// SIMATIC S7-200 project (STEP 7-Micro/WIN), CPU 224 REL 02.01

SYMBOL_TABLE USER1
S1               I0.0
S2               I0.1
S3               I0.2
S4               I0.3
S5               I0.4
S6               I0.5
S7               I0.6
C1S_BW           I1.2     // CY01 S1
C1S_FW           I1.1     // CY01 S2
C2S_UP           I1.0     // CY02 S1
C2S_DWN          I1.3     // CY02 S2
CNV_1            Q1.0
CNV_2            Q1.2
CNV_3            Q1.4
RODLESS          Q0.0
TN_1             Q0.1
TN_2             Q0.6
SUCTION          Q0.2
GRIPPER          Q0.5
CY_1             Q0.3
CY_2             Q0.4
END_SYMBOL_TABLE

ORGANIZATION_BLOCK MAIN:OB1
TITLE=PROGRAM COMMENTS
BEGIN
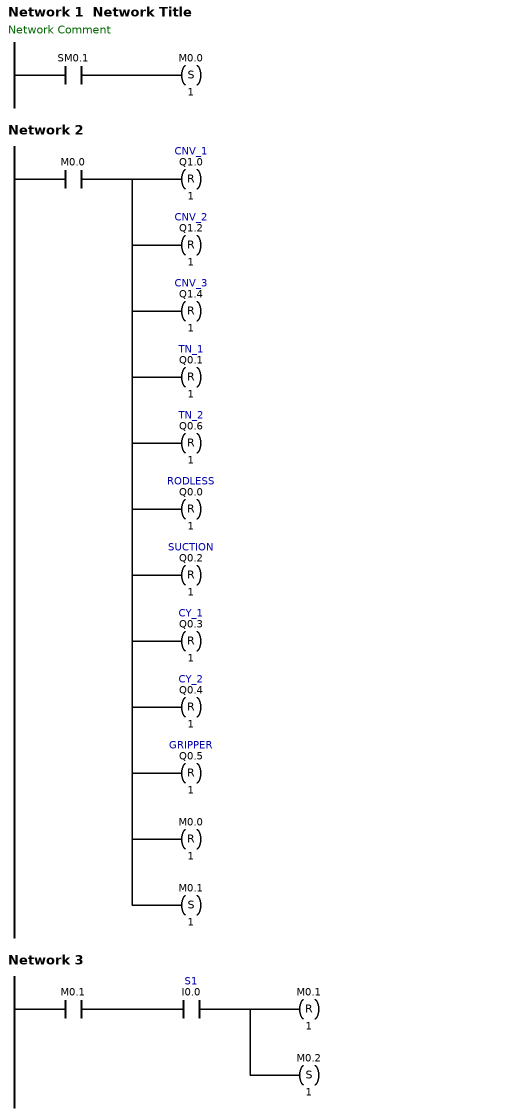
Network 1 // Network Title
// Network Comment
LD     SM0.1
S      M0.0, 1
Network 2
LD     M0.0
R      CNV_1:Q1.0, 1
R      CNV_2:Q1.2, 1
R      CNV_3:Q1.4, 1
R      TN_1:Q0.1, 1
R      TN_2:Q0.6, 1
R      RODLESS:Q0.0, 1
R      SUCTION:Q0.2, 1
R      CY_1:Q0.3, 1
R      CY_2:Q0.4, 1
R      GRIPPER:Q0.5, 1
R      M0.0, 1
S      M0.1, 1
Network 3
LD     M0.1
A      S1:I0.0
R      M0.1, 1
S      M0.2, 1
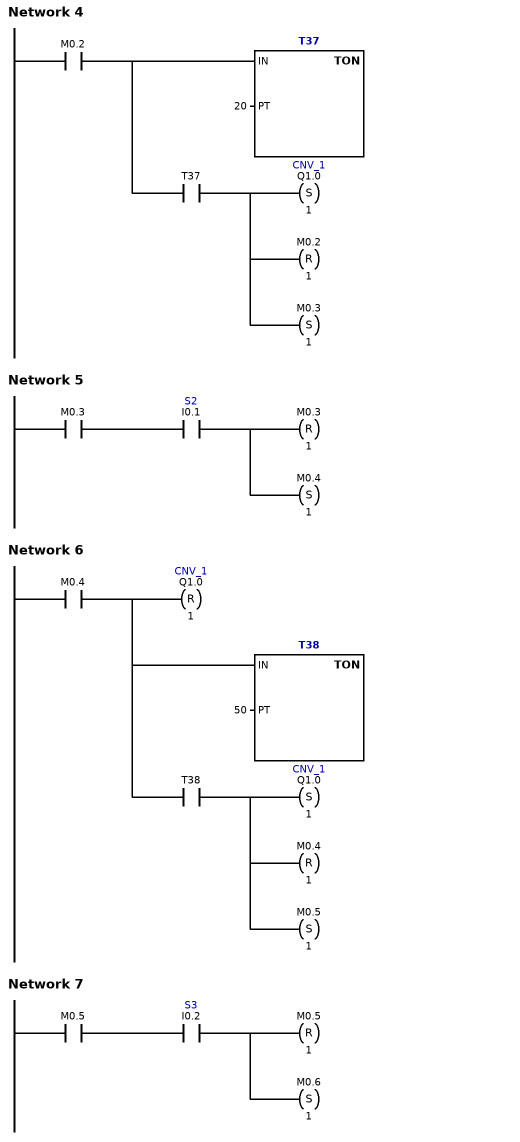
Network 4
LD     M0.2
TON    T37, 20
A      T37
S      CNV_1:Q1.0, 1
R      M0.2, 1
S      M0.3, 1
Network 5
LD     M0.3
A      S2:I0.1
R      M0.3, 1
S      M0.4, 1
Network 6
LD     M0.4
R      CNV_1:Q1.0, 1
TON    T38, 50
A      T38
S      CNV_1:Q1.0, 1
R      M0.4, 1
S      M0.5, 1
Network 7
LD     M0.5
A      S3:I0.2
R      M0.5, 1
S      M0.6, 1
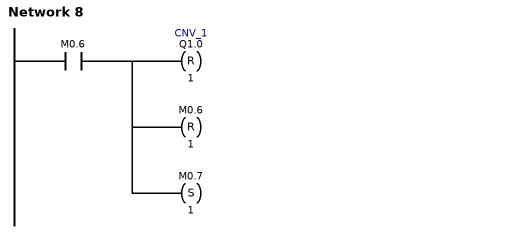
Network 8
LD     M0.6
R      CNV_1:Q1.0, 1
R      M0.6, 1
S      M0.7, 1
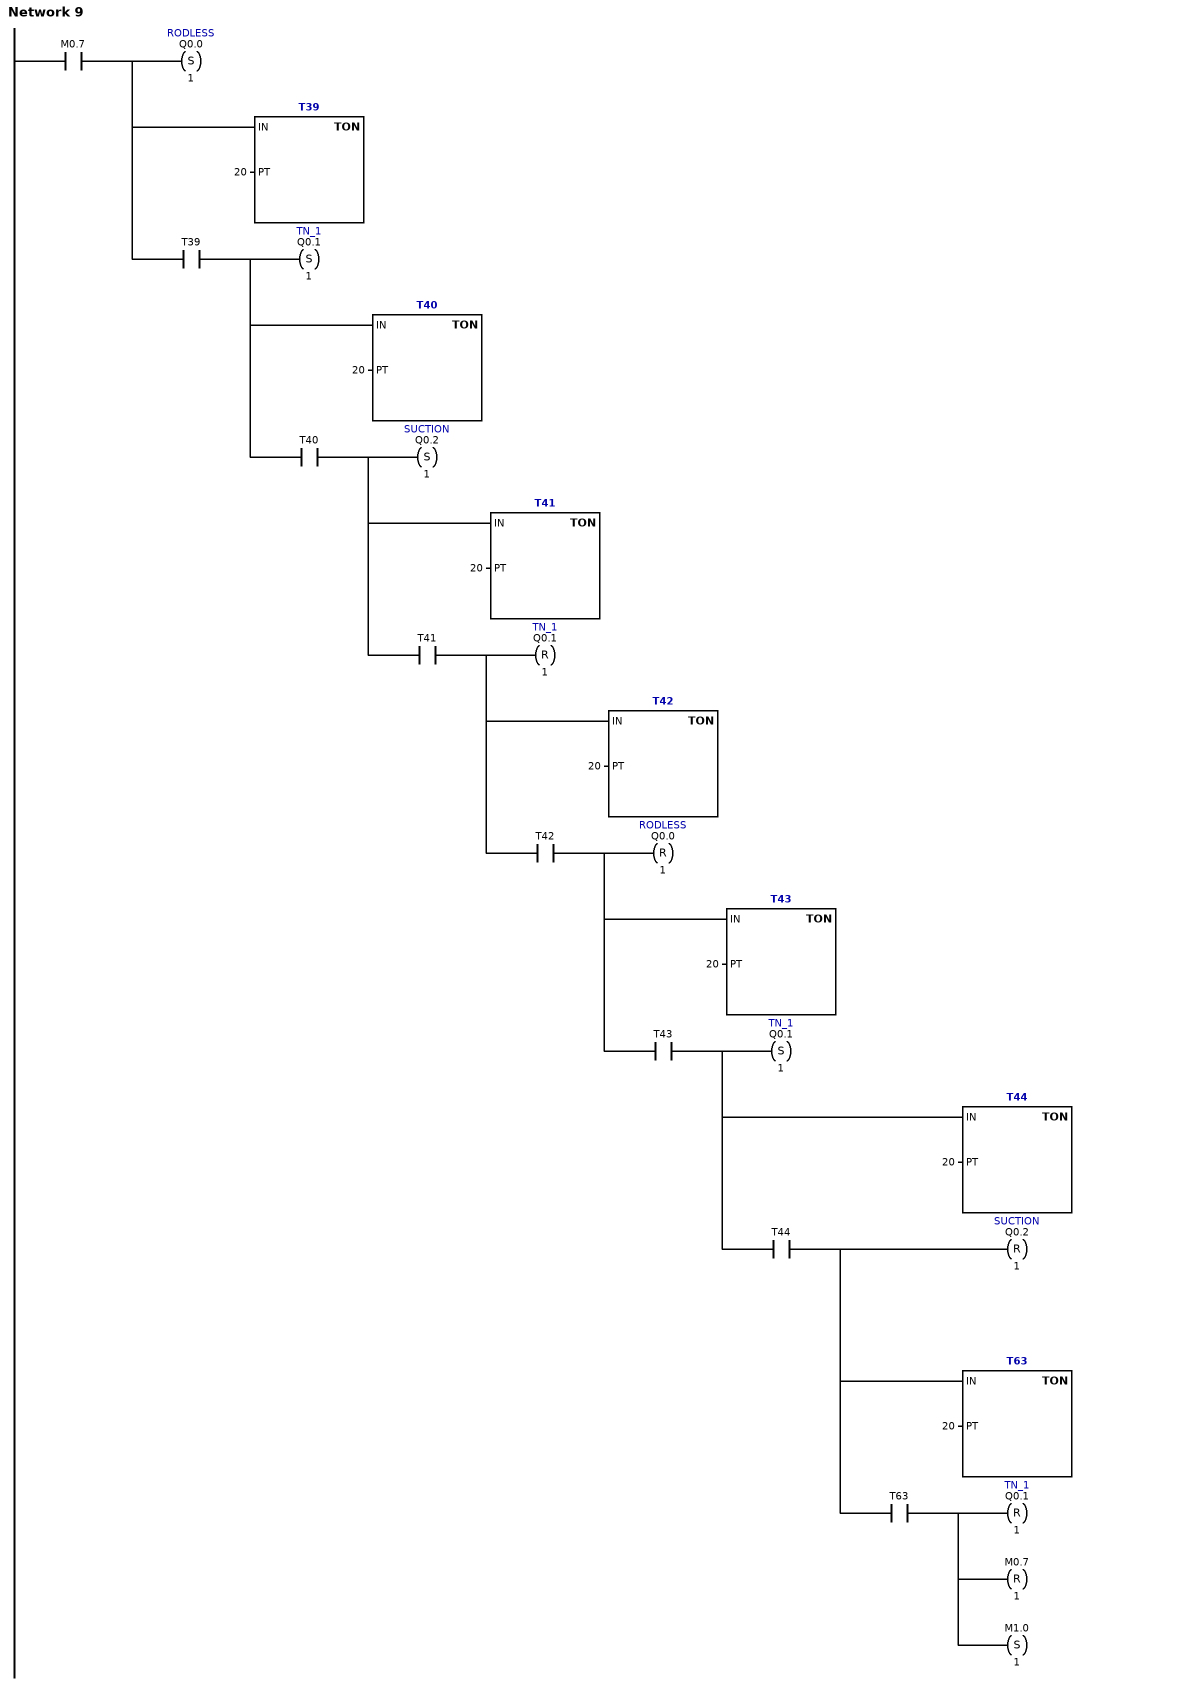
Network 9
// (network saved uncompiled; LAD cells follow)
// row 0: c0 -| |- M0.7 v  c1 -(S) RODLESS:Q0.0, 1
// row 1: c0 ^v  c1 --  c2 [TON T39 IN:=power@row1, PT:=20]
// row 2: c0 ^v  c2 [box]
// row 3: c0 ^  c1 -| |- T39 v  c2 -(S) TN_1:Q0.1, 1
// row 4: c1 ^v  c2 --  c3 [TON T40 IN:=power@row4, PT:=20]
// row 5: c1 ^v  c3 [box]
// row 6: c1 ^  c2 -| |- T40 v  c3 -(S) SUCTION:Q0.2, 1
// row 7: c2 ^v  c3 --  c4 [TON T41 IN:=power@row7, PT:=20]
// row 8: c2 ^v  c4 [box]
// row 9: c2 ^  c3 -| |- T41 v  c4 -(R) TN_1:Q0.1, 1
// row 10: c3 ^v  c4 --  c5 [TON T42 IN:=power@row10, PT:=20]
// row 11: c3 ^v  c5 [box]
// row 12: c3 ^  c4 -| |- T42 v  c5 -(R) RODLESS:Q0.0, 1
// row 13: c4 ^v  c5 --  c6 [TON T43 IN:=power@row13, PT:=20]
// row 14: c4 ^v  c6 [box]
// row 15: c4 ^  c5 -| |- T43 v  c6 -(S) TN_1:Q0.1, 1
// row 16: c5 ^v  c6 --  c7 --  c8 [TON T44 IN:=power@row16, PT:=20]
// row 17: c5 ^v  c8 [box]
// row 18: c5 ^  c6 -| |- T44 v  c7 --  c8 -(R) SUCTION:Q0.2, 1
// row 19: c6 ^v
// row 20: c6 ^v  c7 --  c8 [TON T63 IN:=power@row20, PT:=20]
// row 21: c6 ^v  c8 [box]
// row 22: c6 ^  c7 -| |- T63 v  c8 -(R) TN_1:Q0.1, 1
// row 23: c7 ^v  c8 -(R) M0.7, 1
// row 24: c7 ^  c8 -(S) M1.0, 1
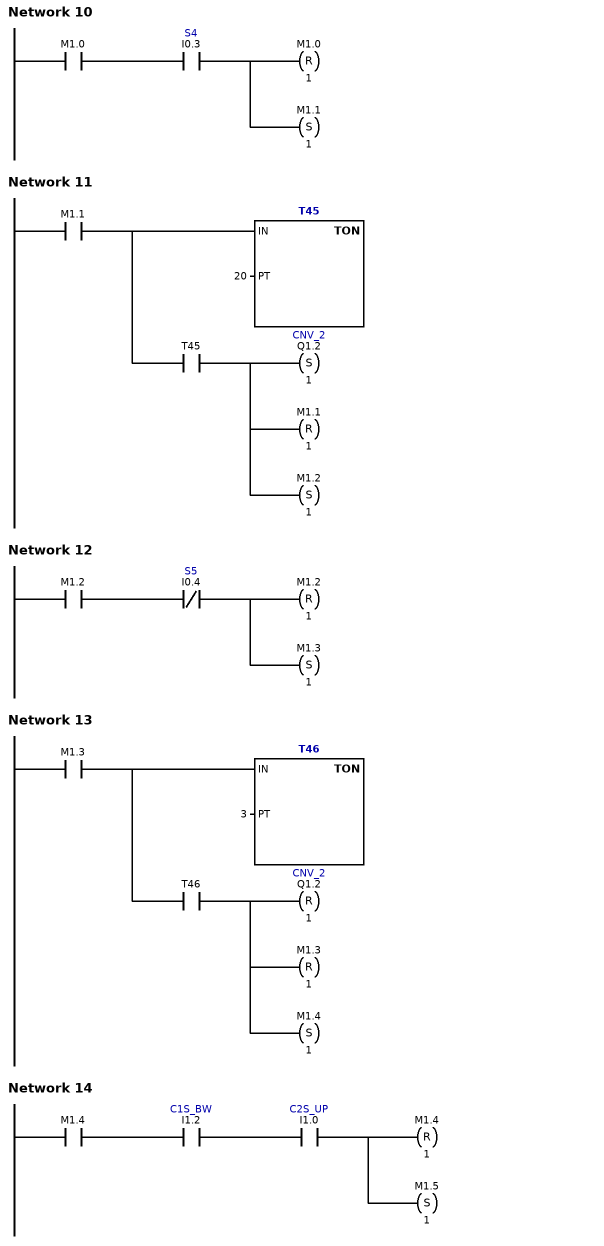
Network 10
LD     M1.0
A      S4:I0.3
R      M1.0, 1
S      M1.1, 1
Network 11
LD     M1.1
TON    T45, 20
A      T45
S      CNV_2:Q1.2, 1
R      M1.1, 1
S      M1.2, 1
Network 12
LD     M1.2
AN     S5:I0.4
R      M1.2, 1
S      M1.3, 1
Network 13
LD     M1.3
TON    T46, 3
A      T46
R      CNV_2:Q1.2, 1
R      M1.3, 1
S      M1.4, 1
Network 14
LD     M1.4
A      C1S_BW:I1.2
A      C2S_UP:I1.0
R      M1.4, 1
S      M1.5, 1
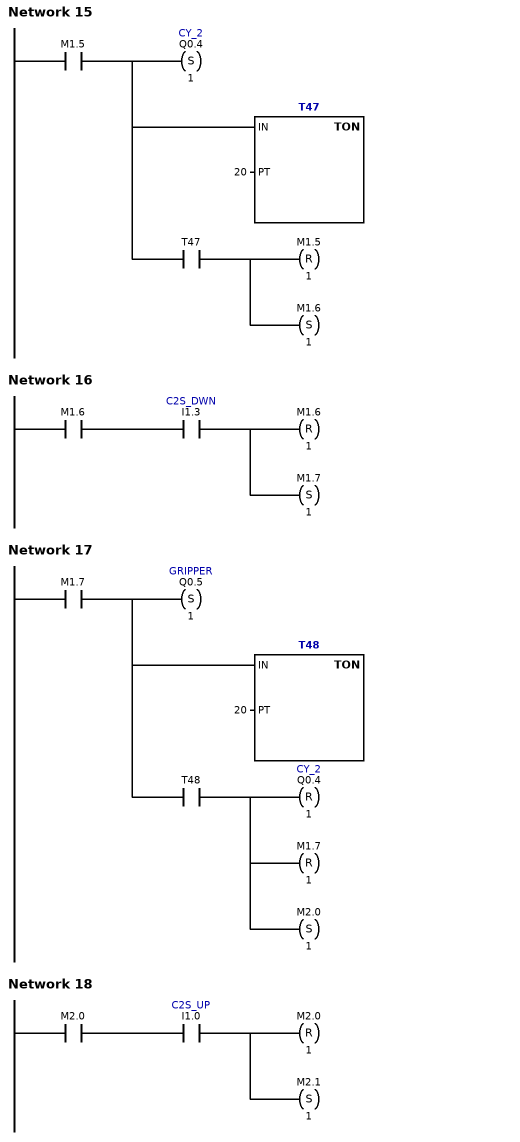
Network 15
LD     M1.5
S      CY_2:Q0.4, 1
TON    T47, 20
A      T47
R      M1.5, 1
S      M1.6, 1
Network 16
LD     M1.6
A      C2S_DWN:I1.3
R      M1.6, 1
S      M1.7, 1
Network 17
LD     M1.7
S      GRIPPER:Q0.5, 1
TON    T48, 20
A      T48
R      CY_2:Q0.4, 1
R      M1.7, 1
S      M2.0, 1
Network 18
LD     M2.0
A      C2S_UP:I1.0
R      M2.0, 1
S      M2.1, 1
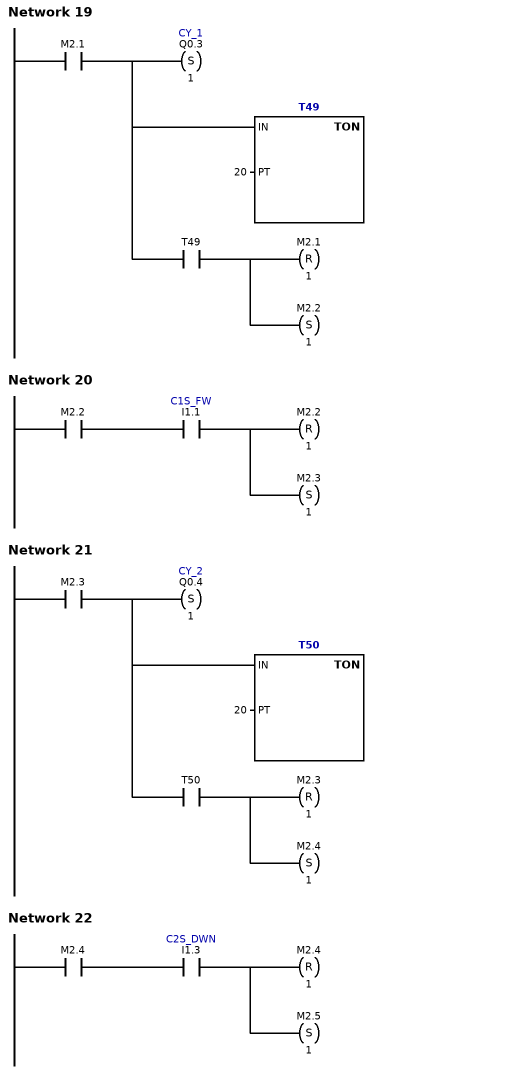
Network 19
LD     M2.1
S      CY_1:Q0.3, 1
TON    T49, 20
A      T49
R      M2.1, 1
S      M2.2, 1
Network 20
// (network saved uncompiled; LAD cells follow)
// row 0: c0 -| |- M2.2  c1 -| |- C1S_FW:I1.1 v  c2 -(R) M2.2, 1
// row 1: c1 ^  c2 -(S) M2.3, 1
Network 21
LD     M2.3
S      CY_2:Q0.4, 1
TON    T50, 20
A      T50
R      M2.3, 1
S      M2.4, 1
Network 22
LD     M2.4
A      C2S_DWN:I1.3
R      M2.4, 1
S      M2.5, 1
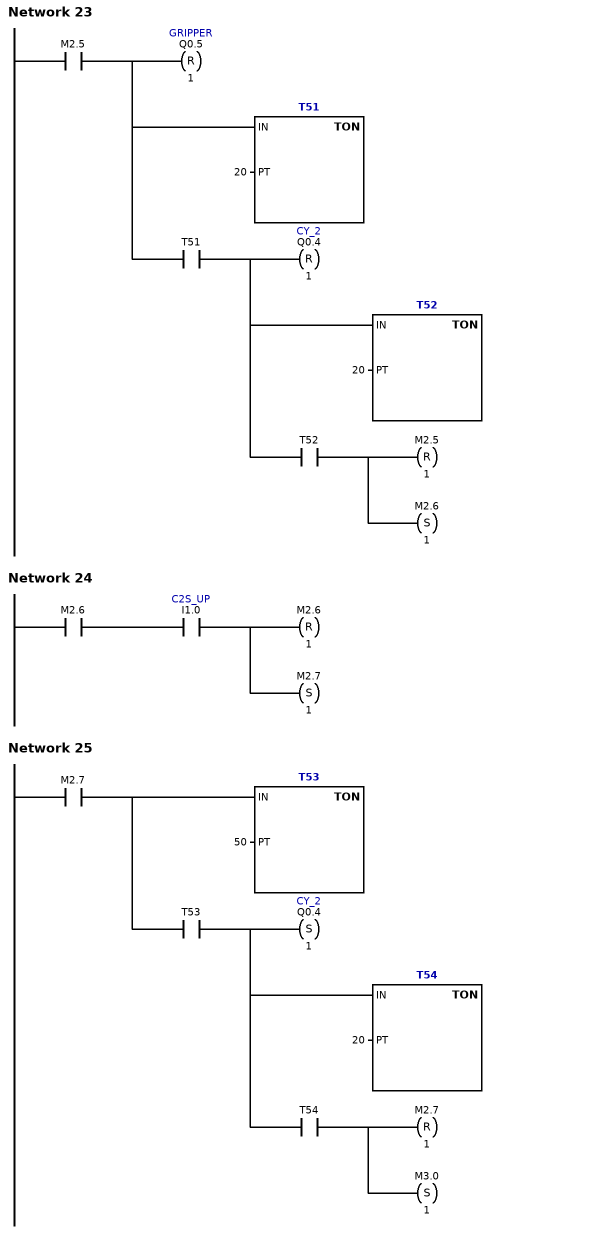
Network 23
LD     M2.5
R      GRIPPER:Q0.5, 1
TON    T51, 20
A      T51
R      CY_2:Q0.4, 1
TON    T52, 20
A      T52
R      M2.5, 1
S      M2.6, 1
Network 24
LD     M2.6
A      C2S_UP:I1.0
R      M2.6, 1
S      M2.7, 1
Network 25
LD     M2.7
TON    T53, 50
A      T53
S      CY_2:Q0.4, 1
TON    T54, 20
A      T54
R      M2.7, 1
S      M3.0, 1
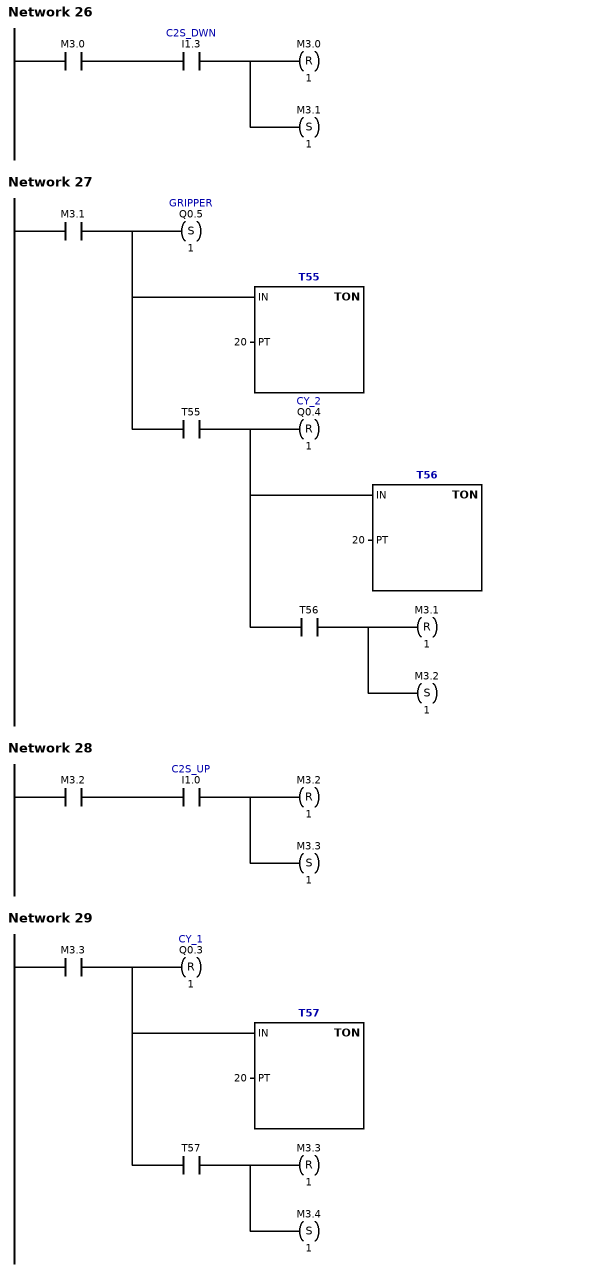
Network 26
LD     M3.0
A      C2S_DWN:I1.3
R      M3.0, 1
S      M3.1, 1
Network 27
LD     M3.1
S      GRIPPER:Q0.5, 1
TON    T55, 20
A      T55
R      CY_2:Q0.4, 1
TON    T56, 20
A      T56
R      M3.1, 1
S      M3.2, 1
Network 28
LD     M3.2
A      C2S_UP:I1.0
R      M3.2, 1
S      M3.3, 1
Network 29
LD     M3.3
R      CY_1:Q0.3, 1
TON    T57, 20
A      T57
R      M3.3, 1
S      M3.4, 1
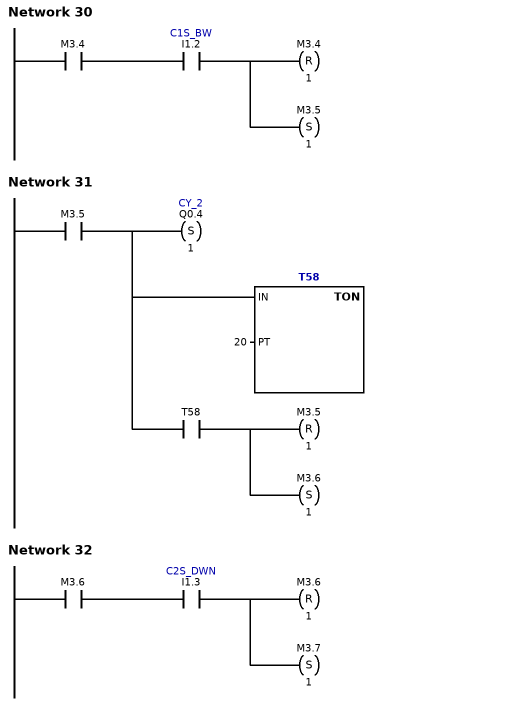
Network 30
// (network saved uncompiled; LAD cells follow)
// row 0: c0 -| |- M3.4  c1 -| |- C1S_BW:I1.2 v  c2 -(R) M3.4, 1
// row 1: c1 ^  c2 -(S) M3.5, 1
Network 31
LD     M3.5
S      CY_2:Q0.4, 1
TON    T58, 20
A      T58
R      M3.5, 1
S      M3.6, 1
Network 32
LD     M3.6
A      C2S_DWN:I1.3
R      M3.6, 1
S      M3.7, 1
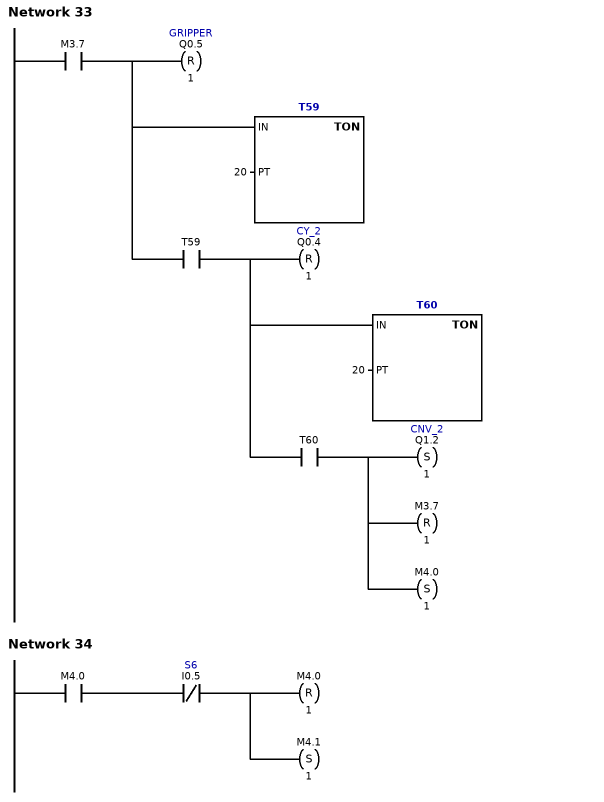
Network 33
LD     M3.7
R      GRIPPER:Q0.5, 1
TON    T59, 20
A      T59
R      CY_2:Q0.4, 1
TON    T60, 20
A      T60
S      CNV_2:Q1.2, 1
R      M3.7, 1
S      M4.0, 1
Network 34
LD     M4.0
AN     S6:I0.5
R      M4.0, 1
S      M4.1, 1
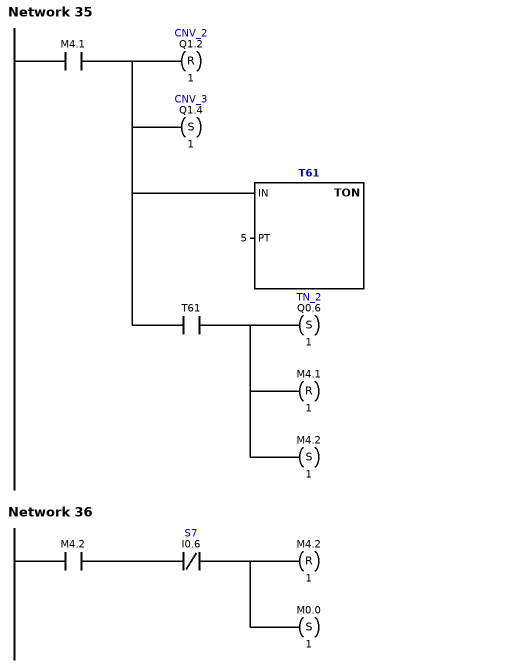
Network 35
// (network saved uncompiled; LAD cells follow)
// row 0: c0 -| |- M4.1 v  c1 -(R) CNV_2:Q1.2, 1
// row 1: c0 ^v  c1 -(S) CNV_3:Q1.4, 1
// row 2: c0 ^v  c1 --  c2 [TON T61 IN:=power@row2, PT:=5]
// row 3: c0 ^v  c2 [box]
// row 4: c0 ^  c1 -| |- T61 v  c2 -(S) TN_2:Q0.6, 1
// row 5: c1 ^v  c2 -(R) M4.1, 1
// row 6: c1 ^  c2 -(S) M4.2, 1
Network 36
LD     M4.2
AN     S7:I0.6
R      M4.2, 1
S      M0.0, 1
END_ORGANIZATION_BLOCK
